TYPE CommandBlocks :
STRUCT

END_STRUCT
END_TYPE

(* stored: Version 1.1.0.1, ProductVersion 3.1.4022.10
   DUT CommandBlocks: Id {44762155-a4ee-4688-ad57-0991b5877603} *)
